// TIA Portal project "2022.06.06_四则运算" (V17)

(* hardware
DEVICE "S7-1200 station_1"  S7-1200 Station
   slot 0: "Rack_0"  S7-1200 Rack  Rack  V1.0
   slot 1: "PLC_1"  CPU 1212C DC/DC/DC  6ES7 212-1AE40-0XB0  V4.5
*)

// ===== PLC "PLC_1"  CPU 1212C DC/DC/DC =====

VAR_GLOBAL   // PLC tag table "默认变量表"
   "Tag_2" AT %MW100 : Word;
   "Tag_3" AT %MW102 : UInt;
   "Tag_4" AT %MW104 : UInt;
   "Tag_5" AT %MW106 : UInt;
   "Tag_6" AT %I0.0 : Bool;
   "Tag_7" AT %M0.0 : Bool;
   "Tag_8" AT %MW10 : Word;
   "Tag_9" AT %MW12 : UInt;
END_VAR

ORGANIZATION_BLOCK "Main"   // OB1, LAD, ProgramCycle
TITLE = "Main Program Sweep (Cycle)"
{ S7_Optimized_Access := 'TRUE' }
VERSION : 0.1
   VAR_INPUT
      Initial_Call : Bool;   // Initial call of this OB
      Remanence : Bool;   // =True, if remanent data are available
   END_VAR
   VAR_TEMP   // added for the SCL form of the ladder/FBD networks
      _w1 : Bool;
   END_VAR
BEGIN

REGION Network 1
   // [(3+5)*30-8]/26
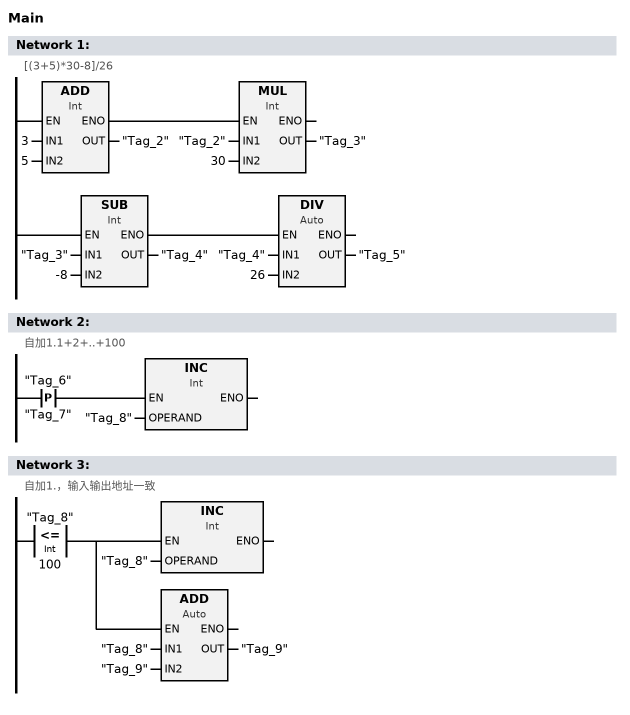
   RUNG wire#powerrail
      { S7_Templates := "SrcType := Int" } Add(in1 := 3, in2 := 5, out => "Tag_2")
      { S7_Templates := "SrcType := Int" } Mul(in1 := "Tag_2", in2 := 30, out => "Tag_3")
   END_RUNG
   RUNG wire#powerrail
      { S7_Templates := "SrcType := Int" } Sub(in1 := "Tag_3", in2 := -8, out => "Tag_4")
      Div(in1 := "Tag_4", in2 := 26, out => "Tag_5")
   END_RUNG
   // the same network as SCL:
   "Tag_2" := 3 + 5;
   "Tag_3" := "Tag_2" * 30;
   "Tag_4" := "Tag_3" - (-8);
   "Tag_5" := "Tag_4" / 26;
END_REGION

REGION Network 2
   // 自加1.1+2+..+100
   RUNG wire#powerrail
      P_Contact(operand := "Tag_6", bit := "Tag_7")
      { S7_Templates := "DestType := Int" } Inc( "Tag_8" )
   END_RUNG
   // the same network as SCL:
   #_w1 := "Tag_6" AND NOT "Tag_7";   // rising edge of "Tag_6"
   "Tag_7" := "Tag_6";
   IF #_w1 THEN "Tag_8" := "Tag_8" + 1; END_IF;
END_REGION

REGION Network 3
   // 自加1.，输入输出地址一致
   RUNG wire#powerrail
      { S7_Templates := "SrcType := Int" } LE_Contact(in1 := "Tag_8", in2 := 100)
      wire#w1
      { S7_Templates := "DestType := Int" } Inc( "Tag_8" )
   END_RUNG
   RUNG wire#w1
      Add(in1 := "Tag_8", in2 := "Tag_9", out => "Tag_9")
   END_RUNG
   // the same network as SCL:
   #_w1 := "Tag_8" <= 100;
   IF #_w1 THEN
       "Tag_8" := "Tag_8" + 1;
       "Tag_9" := "Tag_8" + "Tag_9";
   END_IF;
END_REGION
END_ORGANIZATION_BLOCK